INTERFACE I_AxisStatus

{attribute 'OPC.UA.DA.Property' := '1'}
{attribute 'monitoring':='call'}
PROPERTY LagDistance : LREAL
GET
END_GET
END_PROPERTY

{attribute 'OPC.UA.DA.Property' := '1'}
{attribute 'monitoring':='call'}
PROPERTY MotionState : Tc2_MC2.MC_AxisStates
GET
END_GET
END_PROPERTY

{attribute 'OPC.UA.DA.Property' := '1'}
{attribute 'monitoring':='call'}
PROPERTY SetAcceleration : LREAL
GET
END_GET
END_PROPERTY

{attribute 'OPC.UA.DA.Property' := '1'}
{attribute 'monitoring':='call'}
PROPERTY SetPosition : LREAL
GET
END_GET
END_PROPERTY

{attribute 'OPC.UA.DA.Property' := '1'}
{attribute 'monitoring':='call'}
PROPERTY SetPosModulo : LREAL
GET
END_GET
END_PROPERTY

{attribute 'OPC.UA.DA.Property' := '1'}
{attribute 'monitoring':='call'}
PROPERTY SetVelocity : LREAL
GET
END_GET
END_PROPERTY

END_INTERFACE

(* stored: Version 1.1.0.1, ProductVersion 3.1.4024.12
   Itf I_AxisStatus: Id {0d8e4d9f-bbe7-4022-962a-03340822146e}
   Folder Status: Id {2babc351-48ef-4b6f-81fe-eccd620d0950}
   Folder Dynamics: Id {fc1d2402-8ae3-4cff-8b21-d088c81ee903}
   Property LagDistance: Id {fb0f5634-2c13-0906-1c82-42a6c4a0b8eb}
   Get Get: Id {18961520-ff77-0b09-332d-a95e452e6ec1}
   Property MotionState: Id {9a1b6917-8a35-0e0e-362e-15d08ef85f30}
   Get Get: Id {ceb5f809-7554-0f46-0f5f-29f265091ce7}
   Property SetAcceleration: Id {09f7b76d-4e36-431a-aadf-8b2f5da62ac2}
   Get Get: Id {42e0a9c5-12d2-4bba-b047-7c8e5b06e4e0}
   Property SetPosition: Id {a8587236-2163-4a89-8b5f-70e6cfbe4848}
   Get Get: Id {75e7eacd-60f1-4c7b-a4d3-26f94f884911}
   Property SetPosModulo: Id {075db387-109d-4b7a-8922-b7576e8a327e}
   Get Get: Id {433b8775-c130-4258-bb50-f049217f60f0}
   Property SetVelocity: Id {36c12c75-2ef4-455a-a496-f4f4b70d9ecf}
   Get Get: Id {9564d8da-0709-4fd7-bc5b-a47b2a61ecc8} *)
